Omron CX-Programmer project NewProject (CX-Programmer 9.75)

# PLC NewPLC1: CP1H XA

## Global symbols (name address type ; comment)
0.00 BOOL  ; PB ON
0.01 BOOL  ; PL1
0.02 BOOL  ; PL2
0.03 BOOL  ; PL3
0.04 BOOL  ; PL4
0.05 BOOL  ; SENSOR IN
0.06 BOOL  ; SENSOR OUT
100.00 BOOL  ; SYSTEM ON
100.01 BOOL  ; SYSTEM OFF
100.02 BOOL  ; INDIKATOR LT1
100.03 BOOL  ; INDIKATOR LT2
100.04 BOOL  ; INDIKATOR LT3
100.05 BOOL  ; alarm nyala
101.00 BOOL  ; OPEN
102.00 BOOL  ; orang increment
102.01 BOOL  ; orang decrement
102.03 BOOL  ; orangnya berlebih
102.04 BOOL  ; orangnya cukup
103.00 BOOL  ; alarm nyala
103.01 BOOL  ; OPEN
104.00 BOOL  ; pintu tutup
104.01 BOOL  ; pintu buka
10.01 BOOL  ; LT1
10.02 BOOL  ; LT2
10.03 BOOL  ; LT3
1.00 BOOL  ; PB ON
1.01 BOOL  ; PB OFF
1.04 BOOL  ; Always ON
1.11 BOOL  ; PB BUKA
1.12 BOOL  ; PB TUTUP
2.01 BOOL  ; TOMBOL LT1
2.02 BOOL  ; TOMBOL LT2
2.03 BOOL  ; TOMBOL LT3
590 CHANNEL  ; IN
D1 CHANNEL  ; IN
D2 CHANNEL  ; IN
D3 CHANNEL  ; Maksimal
W10.01 BOOL  ; LT1
W10.02 BOOL  ; LT2
W10.03 BOOL  ; LT3
W10.04 BOOL  ; TURUN
W10.05 BOOL  ; LT2
W10.06 BOOL  ; LT1
W10.07 BOOL  ; LT
W10.08 BOOL  ; END LOOP
W10.09 BOOL  ; END LOOP

## Program NewProgram1 (cyclic task 0)
Local symbols
P_ON BOOL  ; Always ON

### Section Section1
; POWER

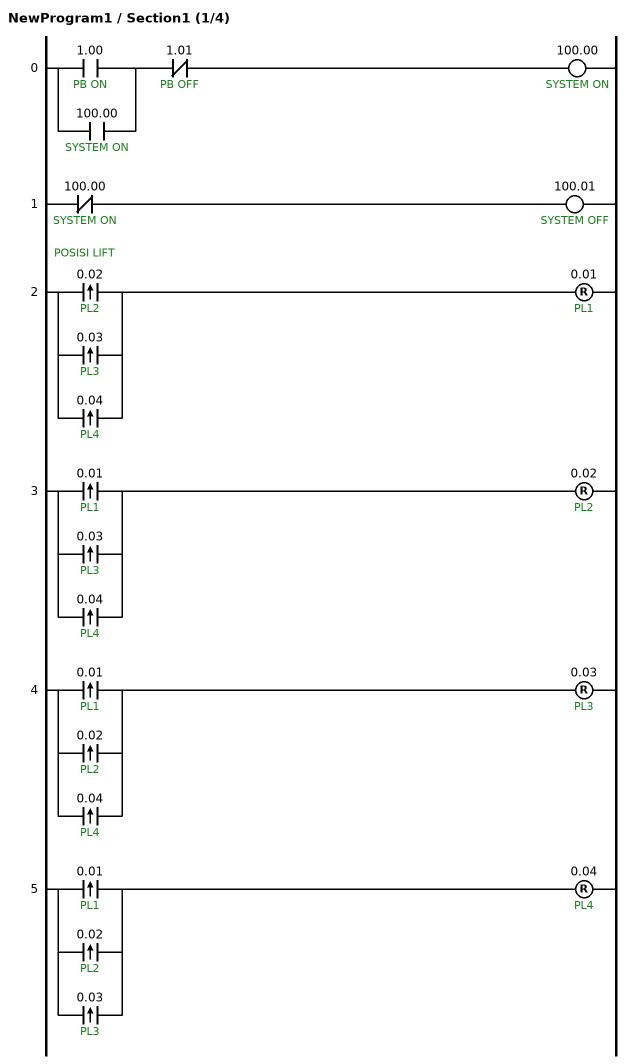
; rung 0
LD 1.00  ; PB ON
OR 100.00  ; SYSTEM ON
ANDNOT 1.01  ; PB OFF
OUT 100.00  ; SYSTEM ON
; rung 1
LDNOT 100.00  ; SYSTEM ON
OUT 100.01  ; SYSTEM OFF
; rung 2: POSISI LIFT
@LD 0.02  ; PL2
@OR 0.03  ; PL3
@OR 0.04  ; PL4
RSET 0.01  ; PL1
; rung 3
@LD 0.01  ; PL1
@OR 0.03  ; PL3
@OR 0.04  ; PL4
RSET 0.02  ; PL2
; rung 4
@LD 0.01  ; PL1
@OR 0.02  ; PL2
@OR 0.04  ; PL4
RSET 0.03  ; PL3
; rung 5
@LD 0.01  ; PL1
@OR 0.02  ; PL2
@OR 0.03  ; PL3
RSET 0.04  ; PL4

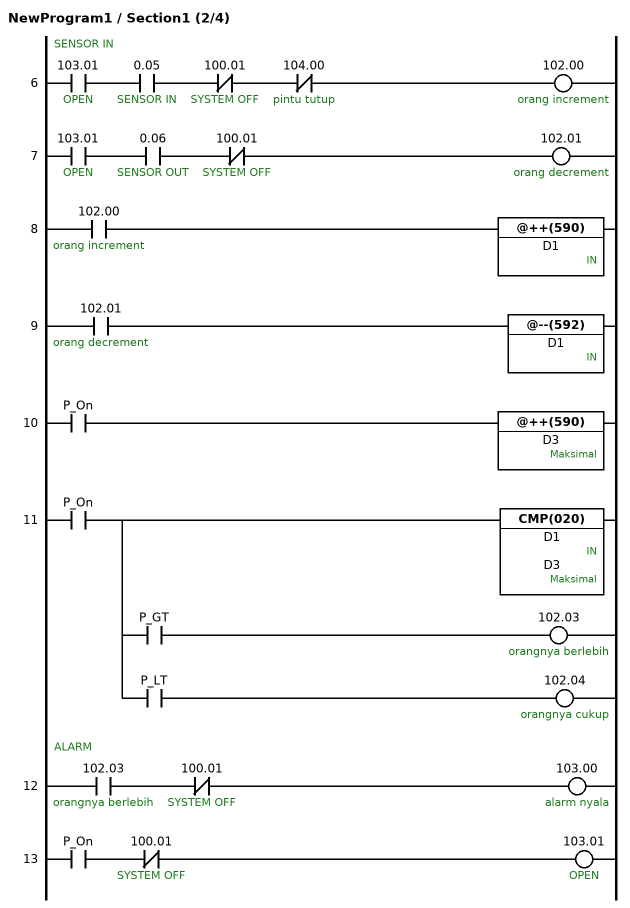
; rung 6: SENSOR IN
LD 103.01  ; OPEN
AND 0.05  ; SENSOR IN
ANDNOT 100.01  ; SYSTEM OFF
ANDNOT 104.00  ; pintu tutup
OUT 102.00  ; orang increment
; rung 7
LD 103.01  ; OPEN
AND 0.06  ; SENSOR OUT
ANDNOT 100.01  ; SYSTEM OFF
OUT 102.01  ; orang decrement
; rung 8
LD 102.00  ; orang increment
@++(590) D1  ; IN
; rung 9
LD 102.01  ; orang decrement
@--(592) D1  ; IN
; rung 10
LD P_On
@++(590) D3  ; Maksimal
; rung 11
LD P_On
OUT TR0
CMP(020) D1 D3  ; IN, Maksimal
AND P_GT
OUT 102.03  ; orangnya berlebih
LD TR0
AND P_LT
OUT 102.04  ; orangnya cukup
; rung 12: ALARM
LD 102.03  ; orangnya berlebih
ANDNOT 100.01  ; SYSTEM OFF
OUT 103.00  ; alarm nyala
; rung 13
LD P_On
ANDNOT 100.01  ; SYSTEM OFF
OUT 103.01  ; OPEN

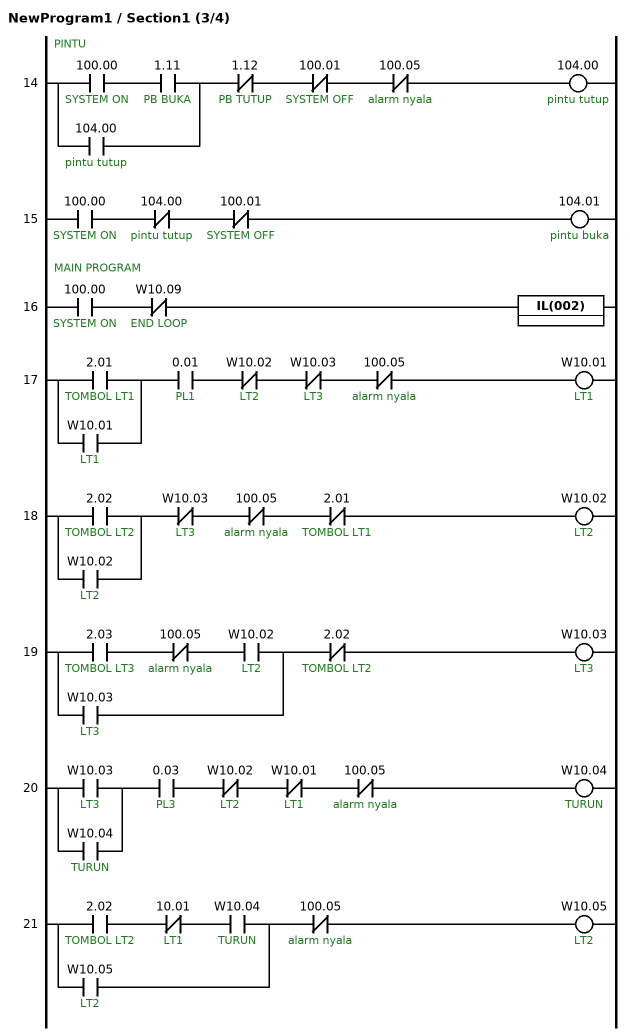
; rung 14: PINTU
LD 100.00  ; SYSTEM ON
AND 1.11  ; PB BUKA
OR 104.00  ; pintu tutup
ANDNOT 1.12  ; PB TUTUP
ANDNOT 100.01  ; SYSTEM OFF
ANDNOT 100.05  ; alarm nyala
OUT 104.00  ; pintu tutup
; rung 15
LD 100.00  ; SYSTEM ON
ANDNOT 104.00  ; pintu tutup
ANDNOT 100.01  ; SYSTEM OFF
OUT 104.01  ; pintu buka
; rung 16: MAIN PROGRAM
LD 100.00  ; SYSTEM ON
ANDNOT W10.09  ; END LOOP
IL(002)
; rung 17
LD 2.01  ; TOMBOL LT1
OR W10.01  ; LT1
AND 0.01  ; PL1
ANDNOT W10.02  ; LT2
ANDNOT W10.03  ; LT3
ANDNOT 100.05  ; alarm nyala
OUT W10.01  ; LT1
; rung 18
LD 2.02  ; TOMBOL LT2
OR W10.02  ; LT2
ANDNOT W10.03  ; LT3
ANDNOT 100.05  ; alarm nyala
ANDNOT 2.01  ; TOMBOL LT1
OUT W10.02  ; LT2
; rung 19
LD 2.03  ; TOMBOL LT3
ANDNOT 100.05  ; alarm nyala
AND W10.02  ; LT2
OR W10.03  ; LT3
ANDNOT 2.02  ; TOMBOL LT2
OUT W10.03  ; LT3
; rung 20
LD W10.03  ; LT3
OR W10.04  ; TURUN
AND 0.03  ; PL3
ANDNOT W10.02  ; LT2
ANDNOT W10.01  ; LT1
ANDNOT 100.05  ; alarm nyala
OUT W10.04  ; TURUN
; rung 21
LD 2.02  ; TOMBOL LT2
ANDNOT 10.01  ; LT1
AND W10.04  ; TURUN
OR W10.05  ; LT2
ANDNOT 100.05  ; alarm nyala
OUT W10.05  ; LT2

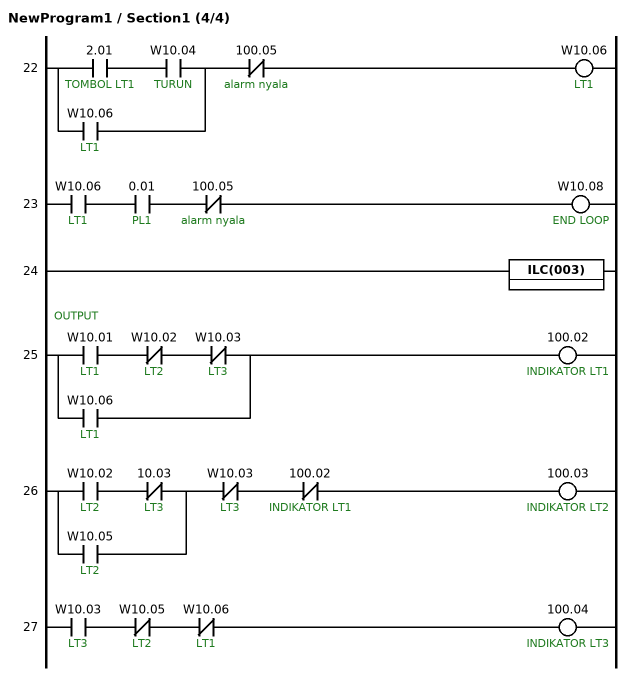
; rung 22
LD 2.01  ; TOMBOL LT1
AND W10.04  ; TURUN
OR W10.06  ; LT1
ANDNOT 100.05  ; alarm nyala
OUT W10.06  ; LT1
; rung 23
LD W10.06  ; LT1
AND 0.01  ; PL1
ANDNOT 100.05  ; alarm nyala
OUT W10.08  ; END LOOP
; rung 24
ILC(003)
; rung 25: OUTPUT
LD W10.01  ; LT1
ANDNOT W10.02  ; LT2
ANDNOT W10.03  ; LT3
OR W10.06  ; LT1
OUT 100.02  ; INDIKATOR LT1
; rung 26
LD W10.02  ; LT2
ANDNOT 10.03  ; LT3
OR W10.05  ; LT2
ANDNOT W10.03  ; LT3
ANDNOT 100.02  ; INDIKATOR LT1
OUT 100.03  ; INDIKATOR LT2
; rung 27
LD W10.03  ; LT3
ANDNOT W10.05  ; LT2
ANDNOT W10.06  ; LT1
OUT 100.04  ; INDIKATOR LT3

### Section END
; rung 0
END(001)